FUNCTION_BLOCK TimeBasedTeach
VAR_INPUT
END_VAR
VAR_OUTPUT
END_VAR
VAR
	bStartTeach	AT%I*	:	BOOL;
	bStopTeach	AT%Q*	:	BOOL;
	
	ton	:	TON;
END_VAR

IF bStartTeach THEN
	ton.IN := NOT ton.Q;
	ton.PT := T#5S;
	
	//ensure StopTeach is False
	bStopTeach := FALSE;
	
	IF ton.Q THEN
		bStartTeach := FALSE;
		bStopTeach := TRUE;
	END_IF
END_IF

END_FUNCTION_BLOCK

(* stored: Version 1.1.0.1, ProductVersion 3.1.4024.12
   POU TimeBasedTeach: Id {88979736-9d2c-4652-8b8c-56b57a98225b}, SpecialFunc None *)
